FUNCTION_BLOCK FB_Observable_INT EXTENDS FB_AbstractObservable
VAR
    _nVal:              INT;
    _nOldVal:           INT;
END_VAR

METHOD FB_init : BOOL
VAR_INPUT
    bInitRetains:       BOOL; // if TRUE, the retain variables are initialized (warm start / cold start)
    bInCopyCode:        BOOL;  // if TRUE, the instance afterwards gets moved into the copy code (online change)
    bAutoNotify:        BOOL;
END_VAR
THIS^._nTypeClass := __SYSTEM.TYPE_CLASS.TYPE_INT;
END_METHOD

PROPERTY nDataSize : UDINT
GET
nDataSize := SIZEOF(INT);
END_GET
END_PROPERTY

PROPERTY nValue16 : INT
GET
nValue16 := THIS^._nVal;
END_GET
SET
THIS^._nOldVal := THIS^._nVal;
THIS^._nVal := nValue16;

THIS^.NotifyWithConditions();
END_SET
END_PROPERTY

PROPERTY PROTECTED pData : POINTER TO BYTE
GET
pData := ADR(THIS^._nVal);
END_GET
END_PROPERTY

METHOD  ValueChanged : BOOL
VAR_INPUT
END_VAR
ValueChanged := THIS^._nOldVal <> THIS^._nVal;
END_METHOD

END_FUNCTION_BLOCK

(* stored: Version 1.1.0.1, ProductVersion 3.1.4024.12
   POU FB_Observable_INT: Id {46000b6a-1bd2-0582-3a83-be6be956a8ad}, SpecialFunc None
   Method FB_init: Id {c85be7ed-de09-036e-2066-6e10af187935}
   Property nDataSize: Id {a84344fa-7a7a-0ae6-2ca6-e285249f4837}
   Get Get: Id {cb25ab96-00d2-0014-1967-47fee7bf9213}
   Property nValue16: Id {7b27de59-b72d-0f7e-369a-e9aa0bb49bd3}
   Get Get: Id {5587f9ef-3a6c-0beb-2ece-9d3636dc689b}
   Set Set: Id {367831f8-8ab7-0f15-2eb4-c683ab052045}
   Property pData: Id {60743575-901b-0665-10f4-d5a55340bf90}
   Get Get: Id {c22eef7a-a8eb-0808-2100-8a461bb311d6}
   Method ValueChanged: Id {026ea014-b221-0f72-1276-b87551885df6} *)
